// TIA Portal V15 SP1 export
// export: Created 2018-01-23T18:59:58.7387467Z, ExportSetting WithDefaults, DisplayName Totally Integrated Automation Portal, DisplayVersion V15 SP1, DisplayName TIA Portal Openness, DisplayVersion V15 SP1, DisplayName TIA Portal Version Control Interface, DisplayVersion V15 SP1, DisplayName Development Version TIA Portal, DisplayVersion V15 SP1, DisplayName STEP 7 Professional, DisplayVersion V15 SP1, DisplayName SIMATIC Energy Suite, DisplayVersion V15 SP1, DisplayName Simocode ES, DisplayVersion V15.1, DisplayName WinCC Professional, DisplayVersion V15 SP1
FUNCTION "Block_1" : Void   // FC1, LAD
{ S7_Optimized_Access := 'TRUE' }
VERSION : 0.1
// stored: AutoNumber true, IsIECCheckEnabled false, SetENOAutomatically False, UDAEnableTagReadback false
BEGIN
END_FUNCTION
